PROGRAM MAIN
VAR
	counter				: UINT;
END_VAR

counter := counter + 1;

PRG_Commands();

END_PROGRAM

(* stored: Version 1.1.0.1, ProductVersion 3.1.4022.10
   POU MAIN: Id {12ac386e-9f2f-456d-9446-322109fb7ee0}, SpecialFunc None *)
